Staubli VAL3: iEmergencyIn.pgx

public program iEmergencyIn(num& nNum[] (dimensions=1))
begin
  nNum=dioGet(iEmergencyIn)
end
